(* PLC project Без имени12.project, Prosoft - Systems Epsilon LD Epsilon LD V1.6.14.0 *)
(* stored: creationDateTime 2021-05-11T13:17:08.4399755, modificationDateTime 2021-05-11T13:16:29.1096554 *)

CONFIGURATION Device
  RESOURCE Application ON PLC
  END_RESOURCE
END_CONFIGURATION
